(* PLC project PackerX.project, CODESYS CODESYS V3.5 SP22 Patch 3 *)
(* stored: creationDateTime 2026-09-23T14:28:37.3474784, modificationDateTime 2026-09-23T14:09:50.4629846 *)

CONFIGURATION Device
END_CONFIGURATION
